FUNCTION_BLOCK FB_LamparaMemorizada_LD
VAR_INPUT
END_VAR
VAR_OUTPUT
END_VAR
VAR
    Lampara AT %Q*: BOOL;
    PulsadorConexion AT %I*: BOOL;
    PulsadorDesconexion AT %I*: BOOL;
    
    Memoria: RS;
END_VAR

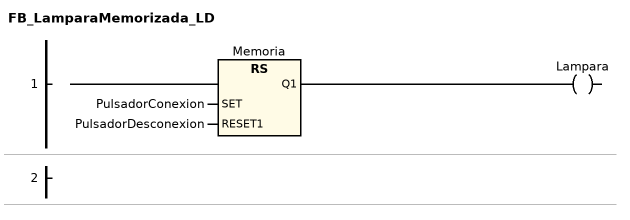
// NETWORK 1
Memoria(SET := PulsadorConexion, RESET1 := PulsadorDesconexion); // RS
Lampara := Memoria.Q1;

// NETWORK 2

END_FUNCTION_BLOCK

(* stored: Version 1.1.0.1, ProductVersion 3.1.4024.12
   POU FB_LamparaMemorizada_LD: Id {3b068606-e4ed-4fff-8c23-37f5b0fb622b}, SpecialFunc None *)
